FUNCTION_BLOCK PUMP_VIEW (* End View of a Rotating Pump *)
  (* Standard: 61499-1 *)
  (* Version 0.1, 2004-09-01, JHC, Rockwell Automation, Deleted QI,QO; set DIA initial value = 0. *)
  (* Version 0.0, 2004-08-30, JHC, Rockwell Automation, Adapted from PUMP_VIEW. *)
  (* Compiler header: package fb.rt.process; *)
  (* Compiler Java Sun JDK 1.4.2 *)
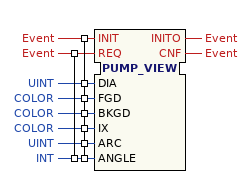
  EVENT_INPUT
    INIT WITH DIA, FGD, BKGD, IX, ARC, ANGLE; (* Initialization *)
    REQ WITH ANGLE; (* Request *)
  END_EVENT
  EVENT_OUTPUT
    INITO; (* Initialization Confirm *)
    CNF; (* Service Confirmation *)
  END_EVENT
  VAR_INPUT
    DIA : UINT; (* Shaft diameter in pixels *)
    FGD : COLOR := COLOR#blue; (* Shaft body color *)
    BKGD : COLOR := COLOR#white; (* Background color *)
    IX : COLOR := COLOR#red; (* Shaft index color *)
    ARC : UINT := 15; (* Shaft mark width *)
    ANGLE : INT; (* Current shaft angle *)
  END_VAR
END_FUNCTION_BLOCK
